{attribute 'linkalways'} 
{attribute 'no_explicit_call' := 'This FB is a CLASS and must be accessed using methods or properties'}
{attribute 'enable_dynamic_creation'}
FUNCTION_BLOCK Node_F_VN_SobelFilterExp EXTENDS VisionNode
VAR
	ipSrcImage : _ITcVnImage;
    ipDestImage : _ITcVnImage;
    eDestDepth : _ETcVnElementType(ETcVnElementType.TCVN_ET_SAME_AS_SOURCE);
    nXOrder : _UDINT(0);
    nYOrder : _UDINT(0);
    nKernelSize : _UDINT(3);
    fScale : _LREAL(1.0);
    fDelta : _LREAL(0.0);
    eBorderType : _ETcVnBorderInterpolationMethod(ETcVnBorderInterpolationMethod.TCVN_BIM_DEFAULT);
    hrPrev : _HRESULT(S_OK);
	hresult : _HRESULT(S_OK);
END_VAR

METHOD PUBLIC  Clone : I_Node
VAR
	pNode : POINTER TO Node_F_VN_SobelFilterExp;
END_VAR
pNode := __NEW(Node_F_VN_SobelFilterExp);
Clone := pNode^;
END_METHOD

METHOD FB_init : BOOL
VAR_INPUT
	bInitRetains : BOOL; // if TRUE, the retain variables are initialized (warm start / cold start)
	bInCopyCode : BOOL;  // if TRUE, the instance afterwards gets moved into the copy code (online change)
END_VAR
AddInput('ipSrcImage', ipSrcImage);
AddParameter('eDestDepth', eDestDepth);
AddParameter('nXOrder', nXOrder);
AddParameter('nYOrder', nYOrder);
AddParameter('nKernelSize', nKernelSize);
AddParameter('fScale', fScale);
AddParameter('fDelta', fDelta);
AddParameter('eBorderType', eBorderType);
AddInput('hrPrev', hrPrev);
AddOutput('ipDestImage', ipDestImage);
AddOutput('hresult',hresult);
END_METHOD

METHOD PROTECTED OnExecute
hresult.Value := F_VN_SobelFilterExp(
	ipSrcImage:= ipSrcImage.Value,
	ipDestImage:= ipDestImage.Value,
	eDestDepth:= eDestDepth.Value,
	nXOrder:= nXOrder.Value,
    nYOrder:= nYOrder.Value,
    nKernelSize:= nKernelSize.Value,
    fScale := fScale.Value,
    fDelta := fDelta.Value,
    eBorderType := eBorderType.Value,
	hrPrev:= hrPrev.Value);
END_METHOD

METHOD PUBLIC PreExecutionCheck
VAR_INPUT
	Check : I_PreExecutionChecks;
END_VAR
VAR
    x_plus_y : UDINT;
END_VAR
Check.IsTrue(ipSrcImage.IsValid, 'ipSrcImage must contain an image');
Check.IsTrue(nKernelSize.IsOdd, 'nKernelSize must be an odd number');
Check.IsTrue((nKernelSize.Value >= 3), 'nKernelSize must be greater than or equal to 3');
Check.IsTrue((nKernelSize.Value <= 31), 'nKernelSize must be less than or equal to 31');

x_plus_y := nXOrder.Value + nYOrder.Value;
Check.IsTrue((x_plus_y > 0), 'nXOrder and nYOrder cannot both be 0');
Check.IsTrue((x_plus_y < nKernelSize.Value), 'nXOrder + nYOrder must be less than nKernelSize');
END_METHOD

END_FUNCTION_BLOCK

(* stored: Version 1.1.0.1, ProductVersion 3.1.4024.15
   POU Node_F_VN_SobelFilterExp: Id {fc22edfd-b73c-0f7a-28b6-452ec7259eab}, SpecialFunc None
   Folder Constructor: Id {96ab34ce-94b5-0d96-1cc3-bd4a3a434684}
   Method Clone: Id {31fd1a5b-24d6-06fd-2c4e-762e140e0ada}
   Method FB_init: Id {3da5fd8c-d23d-00e6-0af3-7b54b99eb17c}
   Method OnExecute: Id {55837029-b84e-08ef-251a-307d2e304d2f}
   Method PreExecutionCheck: Id {9b003d56-0fc5-08b5-3067-c0fcc5c49f2c} *)
